Staubli VAL3: remGetDMOV.pgx

program remGetDMOV(string& sReturn[] (dimensions=1))
  local string sDmov
begin
  // Return whether or not the robot is done moving.
  //
  logMsg("call remGetDMOV")
  if bRemMotionBusy
    sDmov="FALSE"
  else
    sDmov="TRUE"
  endIf
  sReturn="GETDMOV "+sDmov
end
